KUKA KRL program: UP_Service.src, UP_Service.dat

--- UP_Service.src ---
&ACCESS RVO
&REL 7
DEF UP_Service()
  ;=================================================
  ;Unterprogramm Service
  ;Job 6
  ;
  ;=================================================
  ;FOLD Initialisierung
  job = 6
  VZ [Job] = {b FALSE, IDX 0}
  SRC_INIT()
  AuftragStart()
  ;ENDFOLD
  TRIGGER WHEN DISTANCE= 1 DELAY= 0 DO JobNr= Job

  ;Anfahrt
  TRIGGER WHEN DISTANCE= 1 DELAY= 0 DO PosNr= 41
;FOLD PTP Service_VP CONT Vel=50 % PService_VP Tool[15]:Tool_Null Base[15]:base_null;%{PE}
;FOLD Parameters ;%{h}
;Params IlfProvider=kukaroboter.basistech.inlineforms.movement.old; Kuka.IsGlobalPoint=False; Kuka.PointName=Service_VP; Kuka.BlendingEnabled=True; Kuka.MoveDataPtpName=PService_VP; Kuka.VelocityPtp=50; Kuka.CurrentCDSetIndex=0; Kuka.MovementParameterFieldEnabled=True; IlfCommand=PTP
;ENDFOLD
$BWDSTART = FALSE
PDAT_ACT = PPService_VP
FDAT_ACT = FService_VP
BAS(#PTP_PARAMS, 50.0)
SET_CD_PARAMS (0)
PTP XService_VP C_Dis
;ENDFOLD

    ;FOLD FREIGABE_SPS
  ;Warte auf Freigabe von SPS
  Continue
  WAIT_FOR_INPUT_M(eFrg[job].Ef[], TRUE)
  ;Freigabe zyklisch abfragen
  Continue
  Set_CYCFLAG(eFrg[job].Ef[],M_Inbetriebnahme)
  ;ENDFOLD
  ;Eintritt in Stoerbereich an SPS melden
  TRIGGER WHEN DISTANCE= 0 DELAY= 0 DO Reset_(aFrg[job].Ab[]) PRIO= -1

  ;Prozessposition
  TRIGGER WHEN DISTANCE= 1 DELAY= 0 DO PosNr= 45
;FOLD PTP Service_PP Vel=50 % PService_PP Tool[15]:Tool_Null Base[15]:base_null;%{PE}%R 8.5.19,%MKUKATPBASIS,%CMOVE,%VPTP,%P 1:PTP, 2:Service_PP, 3:, 5:50, 7:PService_PP, 9:0
$BWDSTART=FALSE
PDAT_ACT=PPService_PP
FDAT_ACT=FService_PP
BAS(#PTP_PARAMS,50)
SET_CD_PARAMS( 0)
PTP XService_PP
;ENDFOLD

  Handshake(aFrg[job].qEf[],eFrg[job].Ef[],eFrg[job].Pr[])
  ;Serviceposition erreicht
  Handshake(aFrg[job].qPr[],eFrg[job].Pr[],eFrg[job].Rf[],OhneCyc,JobEnde)

  ;Ausfahrt
  ;Austritt aus Stoerbereich an SPS melden
  TRIGGER WHEN DISTANCE= 1 DELAY= 0 DO SetAB(aFrg[job].Ab[]) PRIO=-1

  TRIGGER WHEN DISTANCE= 0 DELAY= 0 DO PosNr= 49
;FOLD PTP Service_NP CONT Vel=50 % PService_NP Tool[15]:Tool_Null Base[15]:base_null;%{PE}
;FOLD Parameters ;%{h}
;Params IlfProvider=kukaroboter.basistech.inlineforms.movement.old; Kuka.IsGlobalPoint=False; Kuka.PointName=Service_NP; Kuka.BlendingEnabled=True; Kuka.MoveDataPtpName=PService_NP; Kuka.VelocityPtp=50; Kuka.CurrentCDSetIndex=0; Kuka.MovementParameterFieldEnabled=True; IlfCommand=PTP
;ENDFOLD
$BWDSTART = FALSE
PDAT_ACT = PPService_NP
FDAT_ACT = FService_NP
BAS(#PTP_PARAMS, 50.0)
SET_CD_PARAMS (0)
PTP XService_NP C_Dis
;ENDFOLD

  CONTINUE
END ;ENDE UP_Service_Program

GLOBAL DEF Rueckzug_Service()
  WHILE PosNr<> 10
    SWITCH PosNr
    CASE 41
      TRIGGER WHEN DISTANCE= 1 DELAY= 0 DO PosNr= 10
      ;MoveParamSet(FDAT, Acc in %, Vel in %, C_PTP in %, C_DIS in mm)
      MoveParamSet(FService_VP,RueckZugAcc,RueckZugVel)
      PTP XService_VP
    CASE 45
      ;Rueckfahrt
      PosNr= 41
    CASE 49
      TRIGGER WHEN DISTANCE= 1 DELAY= 0 DO PosNr= 10
      ;MoveParamSet(FDAT, Acc in %, Vel in %, C_PTP in %, C_DIS in mm)
      MoveParamSet(FService_NP,RueckZugAcc,RueckZugVel)
      PTP XService_NP
    DEFAULT
      LOOP
        ;Falsche PosNr!
        HALT
      ENDLOOP
    ENDSWITCH
  ENDWHILE
  CONTINUE
END ;ENDE Service

--- UP_Service.dat ---
&ACCESS RVO
&REL 7
&PARAM DISKPATH = KRC:\R1\Program\Unterprogramme
DEFDAT  UP_SERVICE
;=================================================
;Unterprogramm Service
;Job 6
;Zelle 6904_ZF_Bin-Picking
;=================================================

INT job

DECL E6POS XService_VP={X -2045.92603,Y -6.20413113,Z 2966.34863,A 179.981964,B 0.0131895663,C -179.960907,S 18,T 10,E1 -3000.00098,E2 0.0,E3 0.0,E4 0.0,E5 0.0,E6 0.0}
DECL FDAT FService_VP={TOOL_NO 15,BASE_NO 15,IPO_FRAME #BASE,POINT2[] " "}
DECL PDAT PPService_VP={VEL 50.0000,ACC 100.000,APO_DIST 50.0000,APO_MODE #CDIS,GEAR_JERK 50.0000,EXAX_IGN 0}
DECL E6POS XService_PP={X -1886.29614,Y -1152.45886,Z 936.626343,A 144.080551,B 0.890194833,C -89.3082886,S 18,T 34,E1 -3000.00098,E2 0.0,E3 0.0,E4 0.0,E5 0.0,E6 0.0}
DECL FDAT FService_PP={TOOL_NO 15,BASE_NO 15,IPO_FRAME #BASE,POINT2[] " ",TQ_STATE FALSE}
DECL PDAT PPService_PP={VEL 100.000,ACC 100.000,APO_DIST 0.0,GEAR_JERK 50.0000,EXAX_IGN 0}
DECL E6POS XService_NP={X -2045.92603,Y -6.20413113,Z 2966.34863,A 179.981964,B 0.0131895663,C -179.960907,S 18,T 10,E1 -3000.00098,E2 0.0,E3 0.0,E4 0.0,E5 0.0,E6 0.0}
DECL FDAT FService_NP={TOOL_NO 15,BASE_NO 15,IPO_FRAME #BASE,POINT2[] " "}
DECL PDAT PPService_NP={VEL 50.0000,ACC 100.000,APO_DIST 50.0000,APO_MODE #CDIS,GEAR_JERK 50.0000,EXAX_IGN 0}

DECL BASIS_SUGG_T LAST_BASIS={POINT1[] "P0                      ",POINT2[] "P0                      ",CP_PARAMS[] "CPDAT0                  ",PTP_PARAMS[] "PDAT0                   ",CONT[] "                        ",CP_VEL[] "2.0                     ",PTP_VEL[] "100                     ",SYNC_PARAMS[] "SYNCDAT                 ",SPL_NAME[] "S0                      ",A_PARAMS[] "ADAT0                   ",PC_SYNCSTRING[] "                        ",GL_SYNCSTRING[] "                        "}
DECL MODULEPARAM_T LAST_TP_PARAMS={PARAMS[] "Kuka.PointName=Service_NP; Kuka.FrameData.base_no=15; Kuka.FrameData.tool_no=15; Kuka.FrameData.ipo_frame=#BASE; Kuka.FrameData.point2=; Kuka.isglobalpoint=False; Kuka.MoveDataPtpName=PService_NP; Kuka.MovementDataPdat.apo_mode=#CDIS; Kuka.MovementDataPdat.apo_dist=50; Kuka.MovementData.vel=50; Kuka.MovementData.acc=100; Kuka.MovementData.exax_ign=0; Kuka.VelocityPtp=50; Kuka.BlendingEnabled=True; Kuka.CurrentCDSetIndex=0    "}
ENDDAT ;ENDE Service
